///////////
// Structure For Inverter. Main Operating Data to be saved ( ex: OPC ) .  
//////////
TYPE INV_Huawei_SL :
STRUCT
	
		MesData				: INV ;  (* INV *) 
	
	// INV Measures
		MesEDay				: REAL ;     	(*/ (kWh) Daily Energy*)
	    MesETot				: REAL ;		(*/ (kWh) Total Energy*)
		MesOn				: BOOL ;        (* Smartlogger is ON*)
		MesI1				: REAL ;        (* (A) AC current phase 1*)
		MesI2				: REAL ;        (* (A) AC current phase 1*)
	    MesI3				: REAL ;        (* (A) AC current phase 1*)
		MesU12				: REAL ;        (*(V) AC Voltage phase1 to phase2*)
        MesU23				: REAL ;        (*(V) AC Voltage phase2 to phase3*)
        MesU31				: REAL ;        (*(V) AC Voltage phase3 to phase1*)
		MesEff				: REAL ; 		(* (%) Inverter efficiency*)
		MesSetptPMax		: REAL ;        (* (kW) Maximal Active power setpoint*)
		MesSetptQMax		: REAL ;        (*(kVAr) Maximal reactive power setpoint*)
		MesSetptQMin		: REAL ;        (*(kVAr) Minimal reactive power setpoint*)
		OUT_SetptPlimit		: REAL ;        (*(kW) Maximal Active power setpoint sent by PPC*)
		OUT_SetptQlimit		: REAL ;        (*(kVAr) Maximal Reactive power setpoint sent by PPC*)

END_STRUCT
END_TYPE

(* stored: Version 1.1.0.1, ProductVersion 3.1.4024.12
   DUT INV_Huawei_SL: Id {75c9e487-2a8d-46da-a7e1-9d0f046aa884} *)
